Staubli VAL3: start.pgx

public program start()
begin
  call InitData()
  call Language()
  call Main()
end
